DATA_BLOCK "FB_AnalogScale_DB"
{ S7_Optimized_Access := 'TRUE' }
VERSION : 0.1
NON_RETAIN
"FB_AnalogScale"

BEGIN

END_DATA_BLOCK

